FUNCTION_BLOCK FB_VirtualCell IMPLEMENTS I_CELL
VAR_INPUT
	
END_VAR
VAR_OUTPUT
END_VAR
VAR
	m_csStateRequest : CELL_ACTION_STATE;
	m_csStateRequestOld : CELL_ACTION_STATE;
	m_csState : CELL_ACTION_STATE;
	m_csStateLastCycle : CELL_ACTION_STATE;
	m_csStateLastAction : CELL_ACTION_STATE;
	
	
	m_csSRWorkingState : CELL_WORKING_STATES := CELL_WORKING_STATES.e_FINISHED;
	m_csSRWorkingStateLast : CELL_WORKING_STATES := CELL_WORKING_STATES.e_FINISHED;
	// Eigenschaften
	m_sName : STRING;
	m_bIsDisassemblyCell : BOOL;
	
	m_iWorkpiece : DINT;
	m_sWorkpieceID : STRING;
	

	m_csCellState : CELL_STATE;
	m_csCellStateLast : CELL_STATE;


	
	m_sErrorString : STRING;
	
	// DataServices
	

	m_sConfigString : STRING;
	m_sConfigStringEndGet : STRING  := '_Get.exe';
	m_sConfigStringEndPut : STRING  := '_Put.exe';
	
	// Virtuelle Zellen Verbindung
	fbVirtualCellIntWriter 	: FB_VirtualCellIntWriter;
	fbJson      			: FB_JsonSaxWriter;
	m_sJsonAction 			: STRING;
	m_sActionPath 			: STRING;
	m_sActionName			: STRING;
	m_sActionPathDir 		: STRING   := 'C:\temp\Actions';
	m_sAMSNetID 			: 	STRING 	:=	'192.168.178.24.1.1';
	
END_VAR

METHOD GetErrorString : STRING
VAR_INPUT
END_VAR
END_METHOD

METHOD GetName : STRING
VAR_INPUT
END_VAR
GetName := m_sName;
END_METHOD

METHOD PUBLIC GetState : INT
VAR_INPUT
	
END_VAR
GetState := CELL_ACTION_STATE.e_Standby;
END_METHOD

METHOD GetWorkpiece : DINT
VAR_INPUT
END_VAR
GetWorkpiece := m_iWorkpiece;
END_METHOD

METHOD IsDisassemblyCell : BOOL
VAR_INPUT
END_VAR
IsDisassemblyCell := FALSE; // Kann keine sein ist virtuell
END_METHOD

METHOD IsError : BOOL
VAR_INPUT
END_VAR
IF m_csCellState = CELL_STATE.e_ERROR THEN
	IsError := TRUE;
END_IF
END_METHOD

METHOD IsIdle : BOOL
VAR_INPUT
END_VAR
IF m_csCellState = CELL_STATE.e_IDEL THEN
	IsIdle := TRUE;
END_IF
END_METHOD

METHOD IsVirtualCell : BOOL
VAR_INPUT
END_VAR
IsVirtualCell :=TRUE;
END_METHOD

METHOD PUBLIC RequestActionState : BOOL
VAR_INPUT
	csStateRequest : CELL_ACTION_STATE;
END_VAR
m_csStateRequest := csStateRequest;
END_METHOD

METHOD RequestWork : BOOL
VAR_INPUT
END_VAR
m_csCellState := CELL_STATE.e_WORKING;
END_METHOD

METHOD SetDisassemblyCell : BOOL
VAR_INPUT
	bIsDisassemblyCell : BOOL;
END_VAR
m_bIsDisassemblyCell := bIsDisassemblyCell;
END_METHOD

METHOD SetGetDataServiceEnable : BOOL
VAR_INPUT
END_VAR

SetGetDataServiceEnable := FALSE;
END_METHOD

METHOD SetName : BOOL
VAR_INPUT
	sName :string ;
END_VAR
m_sName := sName;
END_METHOD

METHOD SetPutDataServiceEnable : BOOL
VAR_INPUT
END_VAR

SetPutDataServiceEnable := FALSE;
END_METHOD

METHOD SetVirtualCell : BOOL
VAR_INPUT
END_VAR
END_METHOD

METHOD SetWorkpiece : BOOL
VAR_INPUT
	iWorkpiece : DINT;
	sWorkpieceID : STRING;
END_VAR
m_iWorkpiece := iWorkpiece;
m_sWorkpieceID := sWorkpieceID;
END_METHOD

METHOD PUBLIC StateMachine : BOOL
VAR_INPUT
END_VAR

//Zellen Zustandsmaschine

CASE m_csCellState OF 
	CELL_STATE.e_IDEL:
			
	
		;
 	CELL_STATE.e_MHS_ACTION;
		//SubRoutine für Aktion beim beladen aktuell leer da keine MHS für eine virtuelle Zelle verfügbar sind 
		;
	CELL_STATE.e_WORKING:
		//SubRoutine zum Durchführen einer Bearbeitung
			//Erstellen des Json-Strings für die Datei		
			fbJson.ResetDocument();
		
			fbJson.StartObject();
            fbJson.AddKey('Name');
			fbJson.AddString(m_sName);
			fbJson.AddKey('WPID');
			fbJson.AddString(m_sWorkpieceID);			
			fbJson.EndObject();
			m_sJsonAction := fbJson.GetDocument();
		
			// Phad der Schnittstellen-Datei
			m_sActionPath := CONCAT (m_sActionPathDir,'\');
			m_sActionPath := CONCAT (m_sActionPath, m_sName);
			m_sActionPath := CONCAT (m_sActionPath, '_');
			m_sActionPath := CONCAT (m_sActionPath, m_sWorkpieceID);
			m_sActionPath := CONCAT (m_sActionPath, '.json');
			
			// Name der Schnittstellen-Datei
			m_sActionName := CONCAT (m_sName, '_');
			m_sActionName := CONCAT (m_sActionName, m_sWorkpieceID);
			m_sActionName := CONCAT (m_sActionName, '.json');
			
			// Nächster Schritt SubRoutine Starten um das Schreiben auszugühren
			IF NOT (CELL_STATE.e_WORKING = m_csCellStateLast) THEN  
				m_csSRWorkingState := CELL_WORKING_STATES.e_START;
			END_IF

			
	CASE m_csSRWorkingState OF
			
			CELL_WORKING_STATES.e_START:
				fbVirtualCellIntWriter.buffRead := m_sJsonAction; // Inhalt der Datei übergeben
				fbVirtualCellIntWriter.sDestPathName := m_sActionPath; // Pfad der Datei
				fbVirtualCellIntWriter.sDestNetId := m_sAMSNetID;// Net Id des HostPC
				fbVirtualCellIntWriter.tTimeOut := DEFAULT_ADS_TIMEOUT;// Fehlerzeit
				fbVirtualCellIntWriter.bExecute := TRUE;// Positive flanke zum Starten
				IF fbVirtualCellIntWriter.bError THEN//
					m_csCellState := CELL_STATE.e_ERROR;
				END_IF

				m_csSRWorkingState := CELL_WORKING_STATES.e_WORKING;

				
			CELL_WORKING_STATES.e_WORKING:	
				fbVirtualCellIntWriter.bExecute := FALSE; // Nur positive Flanke
				IF NOT(fbVirtualCellIntWriter.bBusy) THEN // Der Funktionsblock aufgehört hat zu arbeiten nächster Schritt ggf. das vorhanden sein der Datei prüfen 
					m_csSRWorkingState := CELL_WORKING_STATES.e_FINISHED;
				END_IF
				
			CELL_WORKING_STATES.e_FINISHED:
				m_iWorkpiece := 0;
				m_sWorkpieceID := 'Empty';
				m_csCellState := CELL_STATE.e_IDEL;
			
		END_CASE
		
	CELL_STATE.e_ERROR:
			;
END_CASE

m_csCellStateLast := m_csCellState;
fbVirtualCellIntWriter();
END_METHOD

END_FUNCTION_BLOCK

(* stored: Version 1.1.0.1, ProductVersion 3.1.4024.0
   POU FB_VirtualCell: Id {a90fa4e0-bbd6-44bf-a5e2-a23d2000e0c9}, SpecialFunc None
   Method GetErrorString: Id {ea72647d-72dd-4d26-9c74-65790023a393}
   Method GetName: Id {a4eeaf4b-9099-4090-b5f4-7acfdce5f3b2}
   Method GetState: Id {f76ec9cf-15e5-482f-89cc-03f1c18a1ae9}
   Method GetWorkpiece: Id {deb31da3-968c-468a-a708-ac8b80e8ce29}
   Method IsDisassemblyCell: Id {39df3b55-7f79-4c31-bfee-532f761be0d2}
   Method IsError: Id {2533ada6-4a94-40bd-ad9f-0a03704fa7a8}
   Method IsIdle: Id {2db0ca70-7c53-4c40-a2de-4a0d1f0fff1a}
   Method IsVirtualCell: Id {048bcaad-14c6-4606-994f-088eba23898b}
   Method RequestActionState: Id {575fa3c9-47e2-467f-9657-4296d9f55c66}
   Method RequestWork: Id {c1b7ea6b-aaca-499e-b3a7-02c619a4dd58}
   Method SetDisassemblyCell: Id {ada44e1a-3ad7-44fe-bb6d-8ddcef097431}
   Method SetGetDataServiceEnable: Id {4e8389e7-2bbe-426f-8973-c3019ed534dc}
   Method SetName: Id {27280be0-ca8d-47bb-857a-ad57bc307b63}
   Method SetPutDataServiceEnable: Id {d8340627-f10b-4b6e-9535-3d6fbb7ce993}
   Method SetVirtualCell: Id {93f3f1cb-9ca0-4fe5-9a73-f6e60453fe12}
   Method SetWorkpiece: Id {26bddd69-3d02-467d-b3a6-1c2789da1adf}
   Method StateMachine: Id {75f6fb25-f1c3-49ed-8e42-270cddb5afde} *)
